FUNCTION_BLOCK FEEDERS_HOME_SEQ
VAR_INPUT
END_VAR
VAR_OUTPUT
END_VAR
VAR
END_VAR

END_FUNCTION_BLOCK

(* stored: Version 1.1.0.1, ProductVersion 3.1.4022.18
   POU FEEDERS_HOME_SEQ: Id {2da5084c-3ab1-48e0-8554-c9237a62e0bd}, SpecialFunc None *)
